ABB RAPID module: Module1.modx

MODULE Module1
        PERS tooldata MyTool := [TRUE,[[31.792631019,0,229.638935148],[0.945518576,0,0.325568154,0]],[1,[0,0,1],[1,0,0,0],0,0,0]];
!***********************************************************
    !
    ! Module:  Module1
    !
    ! Description:
    !   <Insert description here>
    !
    ! Author: Student05
    !
    ! Version: 1.0
    !
    !***********************************************************


    !***********************************************************
    !
    ! Procedure main
    !
    !   This is the entry point of your program
    !
    !***********************************************************
    PROC main()
        !Add your code here
    ENDPROC
ENDMODULE
